(* PLC project mtcs_dome, Institute of Astronomy OntoManager 0.0.1 *)
(* stored: creationDateTime 2017-02-07T02:18:52.270690, modificationDateTime 2017-02-07T02:18:52.270690 *)

TYPE DomeParts : STRUCT
  shutter : DomeShutter;  (* Shutter mechanism *)
  rotation : DomeRotation;  (* Rotation mechanism *)
  io : DomeIO;  (* EtherCAT devices *)
  configManager : ConfigManager;  (* The config manager (to load/save/activate configuration data) *)
END_STRUCT;
END_TYPE

TYPE DomeShutterParts : STRUCT
  pumpsRelay : SimpleRelay;  (* Relay to start the pumps motors *)
  upperOpenRelay : SimpleRelay;  (* Relay to open the upper shutter panel *)
  upperCloseRelay : SimpleRelay;  (* Relay to close the upper shutter panel *)
  lowerOpenRelay : SimpleRelay;  (* Relay to open the upper shutter panel *)
  lowerCloseRelay : SimpleRelay;  (* Relay to close the upper shutter panel *)
END_STRUCT;
END_TYPE

TYPE DomeRotationParts : STRUCT
  masterAxis : AngularAxis;  (* Master axis *)
  slaveAxis : AngularAxis;  (* Slave axis *)
  drive : AX52XXDrive;  (* Dual axis drive *)
END_STRUCT;
END_TYPE

TYPE DomeIOParts : STRUCT
  coupler : EtherCatDevice;  (* Coupler *)
  slot1 : EtherCatDevice;  (* Slot 1 *)
  slot2 : EtherCatDevice;  (* Slot 2 *)
  slot3 : EtherCatDevice;  (* Slot 3 *)
  slot4 : EtherCatDevice;  (* Slot 4 *)
  slot5 : EtherCatDevice;  (* Slot 5 *)
  slot6 : EtherCatDevice;  (* Slot 6 *)
  slot7 : EtherCatDevice;  (* Slot 7 *)
  slot8 : EtherCatDevice;  (* Slot 8 *)
END_STRUCT;
END_TYPE

TYPE DomeProcesses : STRUCT
  initialize : Process;  (* Start initializing *)
  lock : Process;  (* Lock the cover *)
  unlock : Process;  (* Unlock the cover *)
  changeOperatingState : ChangeOperatingStateProcess;  (* Change the operating state (e.g. AUTO, MANUAL, ...) *)
  reset : Process;  (* Reset any errors *)
  powerOn : Process;  (* Power on the dome *)
  powerOff : Process;  (* Power off the dome *)
  syncWithAxes : Process;  (* Synchronize the dome once with the axes *)
  trackAxes : Process;  (* Start tracking the axes *)
  stop : Process;  (* Stop the rotation movement and/or tracking *)
END_STRUCT;
END_TYPE

TYPE DomeShutterProcesses : STRUCT
  reset : Process;  (* Reset errors *)
  open : Process;  (* Open both panels *)
  close : Process;  (* Close both panels *)
  stop : Process;  (* Stop the panels *)
  lowerOpen : Process;  (* Open the lower panel *)
  lowerClose : Process;  (* Close the lower panel *)
  upperOpen : Process;  (* Open the upper panel *)
  upperClose : Process;  (* Close the upper panel *)
END_STRUCT;
END_TYPE

TYPE DomeRotationProcesses : STRUCT
  reset : Process;  (* Reset errors *)
  stop : Process;  (* Stop the rotation *)
END_STRUCT;
END_TYPE

TYPE DomeStatuses : STRUCT
  initializationStatus : InitializationStatus;
  healthStatus : HealthStatus;
  busyStatus : BusyStatus;
  operatingStatus : OperatingStatus;
  poweredStatus : PoweredStatus;
END_STRUCT;
END_TYPE

TYPE DomeShutterStatuses : STRUCT
  apertureStatus : ApertureStatus;  (* Combined aperture status (i.e. of both panels) *)
  lowerApertureStatus : ApertureStatus;  (* Aperture status of the lower panel *)
  upperApertureStatus : ApertureStatus;  (* Aperture status of the upper panel *)
  healthStatus : HealthStatus;  (* Health status *)
  busyStatus : BusyStatus;  (* Busy status *)
END_STRUCT;
END_TYPE

TYPE DomeRotationStatuses : STRUCT
  healthStatus : HealthStatus;  (* Health status *)
  busyStatus : BusyStatus;  (* Busy status *)
  poweredStatus : PoweredStatus;  (* Powered status *)
END_STRUCT;
END_TYPE

TYPE DomeIOStatuses : STRUCT
  healthStatus : HealthStatus;  (* Is the I/O in a healthy state? *)
END_STRUCT;
END_TYPE

TYPE DomeConfig : STRUCT
  shutter : DomeShutterConfig;  (* The config of the shutter mechanism *)
  rotation : DomeRotationConfig;  (* The config of the bottom panel set *)
  maxTrackingDistance : LREAL;  (* The maximum distance between telescope and dome while tracking *)
END_STRUCT;
END_TYPE

TYPE DomeShutterConfig : STRUCT
  wirelessPolling : LREAL;  (* Polling frequency of the wireless I/O, in seconds. Negative value = no polling. *)
END_STRUCT;
END_TYPE

TYPE DomeRotationConfig : STRUCT
  maxMasterSlaveLag : LREAL;  (* Below this lag value (in degrees), the lag is considered not an error *)
END_STRUCT;
END_TYPE

FUNCTION_BLOCK SM_Dome
  VAR_INPUT
    {attribute 'OPC.UA.DA' := '1'}
    {attribute 'OPC.UA.DA.Access' := '1'}
    editableConfig : DomeConfig;  (* Editable configuration of the cover *)
  END_VAR
  VAR_OUTPUT
    {attribute 'OPC.UA.DA' := '1'}
    {attribute 'OPC.UA.DA.Access' := '1'}
    actualStatus : STRING;  (* Current status description *)
    previousStatus : STRING;  (* Previous status description *)
    {attribute 'OPC.UA.DA' := '1'}
    {attribute 'OPC.UA.DA.Access' := '1'}
    config : DomeConfig;  (* Active configuration of the cover *)
    {attribute 'OPC.UA.DA' := '1'}
    {attribute 'OPC.UA.DA.Access' := '1'}
    isPoweredOffByPersonInDome : BOOL;  (* True if the dome is powered off due to a person entering the dome *)
    {attribute 'OPC.UA.DA' := '1'}
    {attribute 'OPC.UA.DA.Access' := '1'}
    isTracking : BOOL;  (* True if the dome is tracking the telescope *)
    statuses : DomeStatuses;  (* Statuses of the state machine *)
    parts : DomeParts;  (* Parts of the state machine *)
    processes : DomeProcesses;  (* Processes of the state machine *)
  END_VAR
  VAR_IN_OUT
    {attribute 'OPC.UA.DA' := '0'}
    operatorStatus : OperatorStatus;  (* Reference to the operator (observer/tech) *)
    {attribute 'OPC.UA.DA' := '0'}
    aziPos : AngularPosition;  (* Actual azimuth position of the telescope Axes *)
  END_VAR

            parts.shutter(
    openingAllowed := operatorStatus.tech OR statuses.poweredStatus.enabled,
    initializationStatus := statuses.initializationStatus,
    operatorStatus := operatorStatus,
    operatingStatus := statuses.operatingStatus,
    config := config.shutter);
parts.rotation(
    initializationStatus := statuses.initializationStatus,
    operatorStatus := operatorStatus,
    operatingStatus := statuses.operatingStatus,
    config := config.rotation);
parts.io();
parts.configManager( isEnabled := operatorStatus.tech );
statuses.initializationStatus();
statuses.healthStatus(
    isGood := parts.shutter.statuses.healthStatus.isGood AND (parts.rotation.statuses.healthStatus.isGood AND parts.io.statuses.healthStatus.isGood),
    hasWarning := parts.shutter.statuses.healthStatus.hasWarning OR (parts.rotation.statuses.healthStatus.hasWarning OR parts.io.statuses.healthStatus.hasWarning));
statuses.busyStatus( isBusy := parts.shutter.statuses.busyStatus.busy OR parts.rotation.statuses.busyStatus.busy );
statuses.operatingStatus( superState := statuses.initializationStatus.initialized );
statuses.poweredStatus( isEnabled := parts.rotation.statuses.poweredStatus.enabled );
processes.initialize( isEnabled := statuses.initializationStatus.shutdown OR (statuses.initializationStatus.initializingFailed OR statuses.initializationStatus.initialized) );
processes.lock( isEnabled := operatorStatus.tech AND statuses.initializationStatus.initialized );
processes.unlock( isEnabled := operatorStatus.tech AND statuses.initializationStatus.locked );
processes.changeOperatingState( isEnabled := statuses.busyStatus.idle AND statuses.initializationStatus.initialized );
processes.reset( isEnabled := statuses.busyStatus.idle AND statuses.initializationStatus.initialized );
processes.powerOn( isEnabled := statuses.initializationStatus.initialized AND processes.powerOn.statuses.busyStatus.idle );
processes.powerOff( isEnabled := statuses.initializationStatus.initialized AND processes.powerOff.statuses.busyStatus.idle );
processes.syncWithAxes();
processes.trackAxes( isEnabled := statuses.poweredStatus.enabled );
processes.stop( isEnabled := statuses.busyStatus.busy OR isTracking );

          

{attribute 'TcRpcEnable' := '1'}
METHOD initialize : RequestResults
                  initialize := THIS^.processes.initialize.request();

                
END_METHOD

{attribute 'TcRpcEnable' := '1'}
METHOD lock : RequestResults
                  lock := THIS^.processes.lock.request();

                
END_METHOD

{attribute 'TcRpcEnable' := '1'}
METHOD unlock : RequestResults
                  unlock := THIS^.processes.unlock.request();

                
END_METHOD

{attribute 'TcRpcEnable' := '1'}
METHOD changeOperatingState : RequestResults
  VAR_INPUT
    state : OperatingStates;
  END_VAR
                  changeOperatingState := THIS^.processes.changeOperatingState.request( state := state );

                
END_METHOD

{attribute 'TcRpcEnable' := '1'}
METHOD reset : RequestResults
                  reset := THIS^.processes.reset.request();

                
END_METHOD

{attribute 'TcRpcEnable' := '1'}
METHOD powerOn : RequestResults
                  powerOn := THIS^.processes.powerOn.request();

                
END_METHOD

{attribute 'TcRpcEnable' := '1'}
METHOD powerOff : RequestResults
                  powerOff := THIS^.processes.powerOff.request();

                
END_METHOD

{attribute 'TcRpcEnable' := '1'}
METHOD syncWithAxes : RequestResults
                  syncWithAxes := THIS^.processes.syncWithAxes.request();

                
END_METHOD

{attribute 'TcRpcEnable' := '1'}
METHOD trackAxes : RequestResults
                  trackAxes := THIS^.processes.trackAxes.request();

                
END_METHOD

{attribute 'TcRpcEnable' := '1'}
METHOD stop : RequestResults
                  stop := THIS^.processes.stop.request();

                
END_METHOD

{attribute 'TcRpcEnable' := '1'}
METHOD _log : BOOL
  VAR_INPUT
    name : STRING;  (* Name of this function block instance *)
  END_VAR
  VAR_IN_OUT
    buffer : LogBuffer;  (* Buffer to write all logging to *)
  END_VAR
  VAR
    subBuffer : LogBuffer;  (* Temporary buffer to write logging by parts (sub-statemachines) to *)
  END_VAR
                  THIS^.parts.shutter._log(
    name := 'shutter',
    buffer := subBuffer);
THIS^.parts.rotation._log(
    name := 'rotation',
    buffer := subBuffer);
THIS^.parts.io._log(
    name := 'io',
    buffer := subBuffer);
THIS^.parts.configManager._log(
    name := 'configManager',
    buffer := subBuffer);
LOGGER(
    name := name,
    actualStatus := THIS^.actualStatus,
    previousStatus := THIS^.previousStatus,
    buffer := buffer,
    subBuffer := subBuffer,
    pHealthStatus := ADR(THIS^.statuses.healthStatus),
    pBusyStatus := ADR(THIS^.statuses.busyStatus));

                
END_METHOD
END_FUNCTION_BLOCK

FUNCTION_BLOCK SM_DomeShutter
  VAR_INPUT
    {attribute 'OPC.UA.DA' := '1'}
    {attribute 'OPC.UA.DA.Access' := '1'}
    openingAllowed : BOOL;  (* True if opening is allowed by observer *)
    {attribute 'OPC.UA.DA' := '1'}
    {attribute 'OPC.UA.DA.Access' := '1'}
    lowerOpenSignal : BOOL;  (* False if the signal is not present OR if there is a communication error *)
    {attribute 'OPC.UA.DA' := '1'}
    {attribute 'OPC.UA.DA.Access' := '1'}
    lowerClosedSignal : BOOL;  (* False if the signal is not present OR if there is a communication error *)
    {attribute 'OPC.UA.DA' := '1'}
    {attribute 'OPC.UA.DA.Access' := '1'}
    upperOpenSignal : BOOL;  (* False if the signal is not present OR if there is a communication error *)
    {attribute 'OPC.UA.DA' := '1'}
    {attribute 'OPC.UA.DA.Access' := '1'}
    upperClosedSignal : BOOL;  (* False if the signal is not present OR if there is a communication error *)
    {attribute 'OPC.UA.DA' := '1'}
    {attribute 'OPC.UA.DA.Access' := '1'}
    wirelessTimeout : BOOL;  (* True if the wireless communication to the shutter signals is timing out *)
    {attribute 'OPC.UA.DA' := '1'}
    {attribute 'OPC.UA.DA.Access' := '1'}
    wirelessError : BOOL;  (* True if the wireless communication to the shutter signals is in error (other than timeout) *)
    {attribute 'OPC.UA.DA' := '1'}
    {attribute 'OPC.UA.DA.Access' := '1'}
    wirelessErrorId : UDINT;  (* The error id if wirelessError is true *)
  END_VAR
  VAR_OUTPUT
    {attribute 'OPC.UA.DA' := '1'}
    {attribute 'OPC.UA.DA.Access' := '1'}
    actualStatus : STRING;  (* Current status description *)
    previousStatus : STRING;  (* Previous status description *)
    statuses : DomeShutterStatuses;  (* Statuses of the state machine *)
    parts : DomeShutterParts;  (* Parts of the state machine *)
    processes : DomeShutterProcesses;  (* Processes of the state machine *)
  END_VAR
  VAR_IN_OUT
    {attribute 'OPC.UA.DA' := '0'}
    initializationStatus : InitializationStatus;  (* Dome initialization status (initialized/initializing/...) *)
    {attribute 'OPC.UA.DA' := '0'}
    operatorStatus : OperatorStatus;  (* MTCS operator (observer/tech) *)
    {attribute 'OPC.UA.DA' := '0'}
    operatingStatus : OperatingStatus;  (* Dome operating status (manual/auto) *)
    {attribute 'OPC.UA.DA' := '0'}
    config : DomeShutterConfig;  (* The shutter config *)
  END_VAR

            parts.pumpsRelay( isEnabled := operatorStatus.tech );
parts.upperOpenRelay( isEnabled := operatorStatus.tech );
parts.upperCloseRelay( isEnabled := operatorStatus.tech );
parts.lowerOpenRelay( isEnabled := operatorStatus.tech );
parts.lowerCloseRelay( isEnabled := operatorStatus.tech );
statuses.apertureStatus(
    isOpen := statuses.lowerApertureStatus.open AND statuses.upperApertureStatus.open,
    isClosed := statuses.lowerApertureStatus.closed AND statuses.upperApertureStatus.closed);
statuses.lowerApertureStatus(
    isOpen := lowerOpenSignal,
    isClosed := lowerClosedSignal);
statuses.upperApertureStatus(
    isOpen := upperOpenSignal,
    isClosed := upperClosedSignal);
statuses.healthStatus(
    isGood := (NOT(wirelessTimeout OR wirelessError)) AND (processes.reset.statuses.healthStatus.isGood AND (processes.open.statuses.healthStatus.isGood AND (processes.close.statuses.healthStatus.isGood AND (processes.stop.statuses.healthStatus.isGood AND (processes.lowerOpen.statuses.healthStatus.isGood AND (processes.lowerClose.statuses.healthStatus.isGood AND (processes.upperOpen.statuses.healthStatus.isGood AND processes.upperClose.statuses.healthStatus.isGood))))))),
    hasWarning := processes.reset.statuses.healthStatus.hasWarning OR (processes.open.statuses.healthStatus.hasWarning OR (processes.close.statuses.healthStatus.hasWarning OR (processes.stop.statuses.healthStatus.hasWarning OR (processes.lowerOpen.statuses.healthStatus.hasWarning OR (processes.lowerClose.statuses.healthStatus.hasWarning OR (processes.upperOpen.statuses.healthStatus.hasWarning OR processes.upperClose.statuses.healthStatus.hasWarning)))))));
statuses.busyStatus( isBusy := processes.reset.statuses.busyStatus.busy OR (processes.open.statuses.busyStatus.busy OR (processes.close.statuses.busyStatus.busy OR (processes.stop.statuses.busyStatus.busy OR (processes.lowerOpen.statuses.busyStatus.busy OR (processes.lowerClose.statuses.busyStatus.busy OR (processes.upperOpen.statuses.busyStatus.busy OR processes.upperClose.statuses.busyStatus.busy)))))) );
processes.reset( isEnabled := TRUE );
processes.open( isEnabled := (openingAllowed OR operatorStatus.tech) AND (statuses.busyStatus.idle AND initializationStatus.initialized) );
processes.close( isEnabled := statuses.busyStatus.idle AND initializationStatus.initialized );
processes.stop( isEnabled := statuses.busyStatus.busy );
processes.lowerOpen( isEnabled := processes.open.isEnabled );
processes.lowerClose( isEnabled := processes.close.isEnabled );
processes.upperOpen( isEnabled := processes.close.isEnabled );
processes.upperClose();

          

{attribute 'TcRpcEnable' := '1'}
METHOD reset : RequestResults
                  reset := THIS^.processes.reset.request();

                
END_METHOD

{attribute 'TcRpcEnable' := '1'}
METHOD open : RequestResults
                  open := THIS^.processes.open.request();

                
END_METHOD

{attribute 'TcRpcEnable' := '1'}
METHOD close : RequestResults
                  close := THIS^.processes.close.request();

                
END_METHOD

{attribute 'TcRpcEnable' := '1'}
METHOD stop : RequestResults
                  stop := THIS^.processes.stop.request();

                
END_METHOD

{attribute 'TcRpcEnable' := '1'}
METHOD lowerOpen : RequestResults
                  lowerOpen := THIS^.processes.lowerOpen.request();

                
END_METHOD

{attribute 'TcRpcEnable' := '1'}
METHOD lowerClose : RequestResults
                  lowerClose := THIS^.processes.lowerClose.request();

                
END_METHOD

{attribute 'TcRpcEnable' := '1'}
METHOD upperOpen : RequestResults
                  upperOpen := THIS^.processes.upperOpen.request();

                
END_METHOD

{attribute 'TcRpcEnable' := '1'}
METHOD upperClose : RequestResults
                  upperClose := THIS^.processes.upperClose.request();

                
END_METHOD

{attribute 'TcRpcEnable' := '1'}
METHOD _log : BOOL
  VAR_INPUT
    name : STRING;  (* Name of this function block instance *)
  END_VAR
  VAR_IN_OUT
    buffer : LogBuffer;  (* Buffer to write all logging to *)
  END_VAR
  VAR
    subBuffer : LogBuffer;  (* Temporary buffer to write logging by parts (sub-statemachines) to *)
  END_VAR
                  THIS^.parts.pumpsRelay._log(
    name := 'pumpsRelay',
    buffer := subBuffer);
THIS^.parts.upperOpenRelay._log(
    name := 'upperOpenRelay',
    buffer := subBuffer);
THIS^.parts.upperCloseRelay._log(
    name := 'upperCloseRelay',
    buffer := subBuffer);
THIS^.parts.lowerOpenRelay._log(
    name := 'lowerOpenRelay',
    buffer := subBuffer);
THIS^.parts.lowerCloseRelay._log(
    name := 'lowerCloseRelay',
    buffer := subBuffer);
LOGGER(
    name := name,
    actualStatus := THIS^.actualStatus,
    previousStatus := THIS^.previousStatus,
    buffer := buffer,
    subBuffer := subBuffer,
    pHealthStatus := ADR(THIS^.statuses.healthStatus),
    pBusyStatus := ADR(THIS^.statuses.busyStatus));

                
END_METHOD
END_FUNCTION_BLOCK

FUNCTION_BLOCK SM_DomeRotation
  VAR_OUTPUT
    {attribute 'OPC.UA.DA' := '1'}
    {attribute 'OPC.UA.DA.Access' := '1'}
    actualStatus : STRING;  (* Current status description *)
    previousStatus : STRING;  (* Previous status description *)
    {attribute 'OPC.UA.DA' := '1'}
    {attribute 'OPC.UA.DA.Access' := '1'}
    actPos : AngularPosition;  (* The actual position (same as parts.masterAxis!) *)
    {attribute 'OPC.UA.DA' := '1'}
    {attribute 'OPC.UA.DA.Access' := '1'}
    actVelo : AngularVelocity;  (* The actual velocity (same as parts.masterAxis!) *)
    {attribute 'OPC.UA.DA' := '1'}
    {attribute 'OPC.UA.DA.Access' := '1'}
    actAcc : AngularAcceleration;  (* The actual acceleration (same as parts.masterAxis!) *)
    {attribute 'OPC.UA.DA' := '1'}
    {attribute 'OPC.UA.DA.Access' := '1'}
    actTorqueMaster : Torque;  (* The actual torque on the telescope axis by the master motor *)
    {attribute 'OPC.UA.DA' := '1'}
    {attribute 'OPC.UA.DA.Access' := '1'}
    actTorqueSlave : Torque;  (* The actual torque on the telescope axis by the slave motor *)
    {attribute 'OPC.UA.DA' := '1'}
    {attribute 'OPC.UA.DA.Access' := '1'}
    masterSlaveLag : AngularPosition;  (* masterAxis.actPos - slaveAxis.actPos *)
    {attribute 'OPC.UA.DA' := '1'}
    {attribute 'OPC.UA.DA.Access' := '1'}
    masterSlaveLagError : BOOL;  (* masterSlaveLag >= config.maxMasterSlaveLag *)
    {attribute 'OPC.UA.DA' := '1'}
    {attribute 'OPC.UA.DA.Access' := '1'}
    homingSensorSignal : BOOL;  (* True = at home position *)
    statuses : DomeRotationStatuses;  (* Statuses of the state machine *)
    parts : DomeRotationParts;  (* Parts of the state machine *)
    processes : DomeRotationProcesses;  (* Processes of the state machine *)
  END_VAR
  VAR_IN_OUT
    {attribute 'OPC.UA.DA' := '0'}
    initializationStatus : InitializationStatus;  (* Reference to the MTCS initialization status *)
    {attribute 'OPC.UA.DA' := '0'}
    operatorStatus : OperatorStatus;  (* Reference to the MTCS operator status *)
    {attribute 'OPC.UA.DA' := '0'}
    operatingStatus : OperatingStatus;  (* Reference to the Dome operating status *)
    {attribute 'OPC.UA.DA' := '0'}
    config : DomeRotationConfig;  (* Reference to the rotation config *)
  END_VAR

            parts.masterAxis( isEnabled := operatorStatus.tech );
parts.slaveAxis( isEnabled := operatorStatus.tech );
parts.drive( isEnabled := operatorStatus.tech );
statuses.healthStatus(
    isGood := (parts.masterAxis.statuses.healthStatus.isGood AND (parts.slaveAxis.statuses.healthStatus.isGood AND (parts.drive.statuses.healthStatus.isGood AND (processes.reset.statuses.healthStatus.isGood AND processes.stop.statuses.healthStatus.isGood)))) AND (NOT(masterSlaveLagError)),
    hasWarning := parts.masterAxis.statuses.healthStatus.hasWarning OR (parts.slaveAxis.statuses.healthStatus.hasWarning OR (parts.drive.statuses.healthStatus.hasWarning OR (processes.reset.statuses.healthStatus.hasWarning OR processes.stop.statuses.healthStatus.hasWarning))));
statuses.busyStatus( isBusy := parts.masterAxis.statuses.busyStatus.busy OR (parts.slaveAxis.statuses.busyStatus.busy OR (parts.drive.statuses.busyStatus.busy OR (processes.reset.statuses.busyStatus.busy OR processes.stop.statuses.busyStatus.busy))) );
statuses.poweredStatus( isEnabled := parts.masterAxis.statuses.poweredStatus.enabled AND parts.slaveAxis.statuses.poweredStatus.enabled );
processes.reset( isEnabled := statuses.busyStatus.idle );
processes.stop( isEnabled := statuses.busyStatus.busy );

          

{attribute 'TcRpcEnable' := '1'}
METHOD reset : RequestResults
                  reset := THIS^.processes.reset.request();

                
END_METHOD

{attribute 'TcRpcEnable' := '1'}
METHOD stop : RequestResults
                  stop := THIS^.processes.stop.request();

                
END_METHOD

{attribute 'TcRpcEnable' := '1'}
METHOD _log : BOOL
  VAR_INPUT
    name : STRING;  (* Name of this function block instance *)
  END_VAR
  VAR_IN_OUT
    buffer : LogBuffer;  (* Buffer to write all logging to *)
  END_VAR
  VAR
    subBuffer : LogBuffer;  (* Temporary buffer to write logging by parts (sub-statemachines) to *)
  END_VAR
                  THIS^.parts.masterAxis._log(
    name := 'masterAxis',
    buffer := subBuffer);
THIS^.parts.slaveAxis._log(
    name := 'slaveAxis',
    buffer := subBuffer);
THIS^.parts.drive._log(
    name := 'drive',
    buffer := subBuffer);
LOGGER(
    name := name,
    actualStatus := THIS^.actualStatus,
    previousStatus := THIS^.previousStatus,
    buffer := buffer,
    subBuffer := subBuffer,
    pHealthStatus := ADR(THIS^.statuses.healthStatus),
    pBusyStatus := ADR(THIS^.statuses.busyStatus));

                
END_METHOD
END_FUNCTION_BLOCK

FUNCTION_BLOCK SM_DomeIO
  VAR_OUTPUT
    {attribute 'OPC.UA.DA' := '1'}
    {attribute 'OPC.UA.DA.Access' := '1'}
    actualStatus : STRING;  (* Current status description *)
    previousStatus : STRING;  (* Previous status description *)
    statuses : DomeIOStatuses;  (* Statuses of the state machine *)
    parts : DomeIOParts;  (* Parts of the state machine *)
  END_VAR

            parts.coupler(
    id := '110A1',
    typeId := 'EK1101');
parts.slot1(
    id := '115A1',
    typeId := 'EL2008');
parts.slot2(
    id := '116A1',
    typeId := 'EL4008');
parts.slot3(
    id := '117A1',
    typeId := 'EL1088');
parts.slot4(
    id := '118A1',
    typeId := 'EL5002');
parts.slot5(
    id := '118A5',
    typeId := 'EL5002');
parts.slot6(
    id := '119A1',
    typeId := 'EL5002');
parts.slot7(
    id := '119A5',
    typeId := 'EL5002');
parts.slot8(
    id := '111A1',
    typeId := 'EL2622');
statuses.healthStatus( isGood := parts.coupler.statuses.healthStatus.isGood AND (parts.slot1.statuses.healthStatus.isGood AND (parts.slot2.statuses.healthStatus.isGood AND (parts.slot3.statuses.healthStatus.isGood AND (parts.slot4.statuses.healthStatus.isGood AND (parts.slot5.statuses.healthStatus.isGood AND (parts.slot6.statuses.healthStatus.isGood AND (parts.slot7.statuses.healthStatus.isGood AND parts.slot8.statuses.healthStatus.isGood))))))) );

          

{attribute 'TcRpcEnable' := '1'}
METHOD _log : BOOL
  VAR_INPUT
    name : STRING;  (* Name of this function block instance *)
  END_VAR
  VAR_IN_OUT
    buffer : LogBuffer;  (* Buffer to write all logging to *)
  END_VAR
  VAR
    subBuffer : LogBuffer;  (* Temporary buffer to write logging by parts (sub-statemachines) to *)
  END_VAR
                  THIS^.parts.coupler._log(
    name := 'coupler',
    buffer := subBuffer);
THIS^.parts.slot1._log(
    name := 'slot1',
    buffer := subBuffer);
THIS^.parts.slot2._log(
    name := 'slot2',
    buffer := subBuffer);
THIS^.parts.slot3._log(
    name := 'slot3',
    buffer := subBuffer);
THIS^.parts.slot4._log(
    name := 'slot4',
    buffer := subBuffer);
THIS^.parts.slot5._log(
    name := 'slot5',
    buffer := subBuffer);
THIS^.parts.slot6._log(
    name := 'slot6',
    buffer := subBuffer);
THIS^.parts.slot7._log(
    name := 'slot7',
    buffer := subBuffer);
THIS^.parts.slot8._log(
    name := 'slot8',
    buffer := subBuffer);
LOGGER(
    name := name,
    actualStatus := THIS^.actualStatus,
    previousStatus := THIS^.previousStatus,
    buffer := buffer,
    subBuffer := subBuffer,
    pHealthStatus := ADR(THIS^.statuses.healthStatus));

                
END_METHOD
END_FUNCTION_BLOCK
